(* CODESYS project ObjectOrientedProgramming.project
   Author: Manfred Werner
   Description: This example shows how OOP could be used to simplify the implementation of the management of different types of rooms.
      Start reading with the Interaces followed by the POU Building Manager.
   Title: Object Oriented Programming

Project tree, tasks and I/O mapping:
  Device : CODESYS Control Win V3 x64, 3S - Smart Software Solutions GmbH, version 3.5.15.0
    application BuildingApplication
      libraries: Util, 3.4.1.20 (System); Standard, * (System); CmpBitmapPool, * (System)
      task BuildingTask (cyclic, interval t#50ms, priority 1) calls BuildingManager
      Building_Objects/
        RoomFBs/
          function block RoomType3 [ST]: Operation_Daytime, SetTemperature, Operation_Nighttime, GetTemperature
          function block Roomtype1 [ST]: Operation_Daytime, SetLight, GetLight, Operation_Nighttime
          function block RoomType2 [ST]: SetLight
        function block CheckFB [CFC]
        Visualizations/
          visualisation Bulb
          visualisation Building
        global variables GlobalConstants
        program BuildingManager [ST]
        Interfaces/
          interface ITemp: SetTemperature, GetTemperature
          interface ILight: GetLight, SetLight
          interface IRoom: Operation_Nighttime, Operation_Daytime
      image pool ImagePool
      license
  libraries: VisuSymbols, 3.5.10.0 (System)
  text list GlobalTextList
  5ce3da45-db07-42e7-a21c-a00fff4ed8f6|C:\Users\a.werner\Documents\background.jpg
  00000000-0000-0000-0000-000000000000|C:\Users\m.lamp\Documents\license.txt
*)

// Device/BuildingApplication/Building_Objects/GlobalConstants
VAR_GLOBAL CONSTANT
	iNumberOfRooms:INT:=8;
END_VAR

// Device/BuildingApplication/Building_Objects/BuildingManager
PROGRAM BuildingManager
VAR
	(* define all rooms *)
	r1:RoomType1;		
	r2:RoomType3;
	r3:RoomType2;
	r4:RoomType3;
	r5:RoomType1;
	r6:RoomType3;
	r7:RoomType2;
	r8:RoomType1;
	(* Array of rooms simpilifies working with the building.*)
	Rooms: ARRAY [1..iNumberOfRooms] OF IRoom:=[r1,r2,r3,r4,r5,r6,r7,r8];
	CheckTimeOfDay: CheckFB; 	(* It's getting day? It's getting night? *)		
	xDusk: BOOL; (* nighttime *)
	xDawn:BOOL; (* daytime*)
	itfTemp: ITemp;
	xTemp: BOOL; (* Result of the Interface mapping.*) 
	i: INT;
END_VAR

(* Check if there is daytime or nighttime.*)
CheckTimeOfDay(xGetsDay=>xDawn,xGetsNight=>xDusk);
FOR i:=1 TO iNumberOfRooms DO
	IF xDawn THEN	(* Daytime*)
		Rooms[i].Operation_Daytime(); (* Disable the light and depending on the roomtype set the temperature. *)
	END_IF
	IF xDusk THEN	(* Nighttime *)
		Rooms[i].Operation_Nighttime(); (* Enable the light and depending on the roomtype set the temperature. *)
	END_IF
	
	(* If temperature is available for the Room, then set the temperature  --> RoomType3*)
	xTemp:=__QUERYINTERFACE(Rooms[i], itfTemp);
	IF xTemp AND i=6 THEN
		(* Now itfTemp has the address of Rooms[6] *)
		itfTemp.SetTemperature(35); (* The temperature of the Rooms[6] is set. *)
	END_IF
	
END_FOR

END_PROGRAM

// Device/BuildingApplication/Building_Objects/RoomFBs/RoomType3
(* Extended Room with an extra light and temperature. *)
FUNCTION_BLOCK RoomType3 EXTENDS Roomtype2 IMPLEMENTS ITemp
VAR_INPUT
END_VAR
VAR_OUTPUT
END_VAR
VAR
	iTemperature:INT;
END_VAR

(* This method overrides the inherited Operation_Daytime method from RoomType2. *)
METHOD Operation_Daytime : BOOL
VAR_INPUT
END_VAR
VAR
END_VAR
SUPER^.Operation_Daytime(); (* Disables the light.*)
SetTemperature(25); (* Additionally the temperature is set *)
END_METHOD

(* Implementation of the ITemp Interface *)
METHOD SetTemperature : BOOL
VAR_INPUT
	iNewTemperature:INT;
END_VAR
VAR
END_VAR
(* New temperature is set *)
iTemperature:=iNewTemperature;
END_METHOD

(* This method overrides the inherrited Operation_Nighttime method from RoomType2. *)
METHOD Operation_Nighttime : BOOL
VAR_INPUT
END_VAR
VAR
END_VAR
SUPER^.Operation_Nighttime(); (* Enables the light.*)
SetTemperature(15); (* Additionally the temperature is set *)
END_METHOD

(* Implementation of the ITemp Interface *)
METHOD GetTemperature : INT
VAR_INPUT
END_VAR
VAR
END_VAR
(* Get the temperature *)
GetTemperature:=iTemperature;
END_METHOD

END_FUNCTION_BLOCK

// Device/BuildingApplication/Building_Objects/RoomFBs/RoomType2
(* Extended Room with an extra light *)
FUNCTION_BLOCK RoomType2 EXTENDS Roomtype1
VAR_INPUT
END_VAR
VAR_OUTPUT
END_VAR
VAR
	bAdditionalLight:BOOL;
END_VAR

(* This method overrides the inherited SetLight method from RoomType1. *)
METHOD SetLight : BOOL
VAR_INPUT
	b:BOOL;
END_VAR
VAR
END_VAR
SUPER^.SetLight(b); (* Call the inherrited mehtod *)(* equal bLight:=b; *)
bAdditionalLight:=b;
END_METHOD

END_FUNCTION_BLOCK

// Device/BuildingApplication/Building_Objects/RoomFBs/Roomtype1
(* Simple room with only one light. *)	
FUNCTION_BLOCK Roomtype1 IMPLEMENTS IRoom, ILight
VAR_INPUT
END_VAR
VAR_OUTPUT
END_VAR
VAR
	bLight:BOOL;
END_VAR

(* Implementation of the IRoom Interface *)
METHOD Operation_Daytime : BOOL
VAR_INPUT
END_VAR
VAR
END_VAR
SetLight(FALSE); (* Disables the light *)
END_METHOD

(* Implementation of the ILight Interface *)
METHOD SetLight : BOOL
VAR_INPUT
	b:BOOL;
END_VAR
VAR
END_VAR
(* Set a new light value *)
bLight:=b;
END_METHOD

(* Implementation of the ILight Interface *)
METHOD GetLight : BOOL
VAR_INPUT
END_VAR
VAR
END_VAR
(* Returns the value of the light. *)
GetLight:=bLight;
END_METHOD

(* Implementation of the IRoom Interface *)
METHOD Operation_Nighttime : BOOL
VAR_INPUT
END_VAR
VAR
END_VAR
SetLight(TRUE); (* Enables the light *)
END_METHOD

END_FUNCTION_BLOCK

// Device/BuildingApplication/Building_Objects/Interfaces/IRoom
INTERFACE IRoom EXTENDS __system.IQueryInterface

METHOD Operation_Nighttime : BOOL
VAR_INPUT
END_VAR
VAR
END_VAR
END_METHOD

METHOD Operation_Daytime : BOOL
VAR_INPUT
END_VAR
VAR
END_VAR
END_METHOD

END_INTERFACE

// Device/BuildingApplication/Building_Objects/Interfaces/ILight
INTERFACE ILight

METHOD GetLight : BOOL
VAR_INPUT
END_VAR
VAR
END_VAR
END_METHOD

METHOD SetLight : BOOL
VAR_INPUT
	b:BOOL;
END_VAR
VAR
END_VAR
END_METHOD

END_INTERFACE

// Device/BuildingApplication/Building_Objects/Interfaces/ITemp
INTERFACE ITemp

METHOD SetTemperature : BOOL
VAR_INPUT
	iNewTemperature:INT;
END_VAR
VAR
END_VAR
END_METHOD

METHOD GetTemperature : INT
VAR_INPUT
END_VAR
VAR
END_VAR
END_METHOD

END_INTERFACE

// Device/BuildingApplication/Building_Objects/CheckFB
FUNCTION_BLOCK CheckFB
VAR_INPUT
END_VAR
VAR_OUTPUT
	xGetsNight:BOOL;
	xGetsDay:BOOL;
END_VAR
VAR
	blinking: BLINK;
	DayTrigger: R_TRIG;
	NightTrigger: F_TRIG;
END_VAR

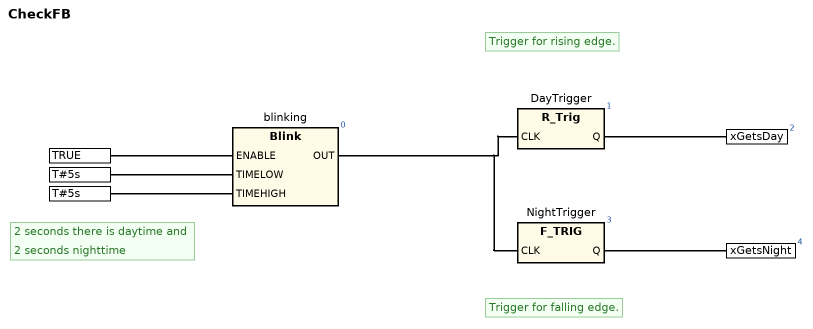
blinking(ENABLE := TRUE, TIMELOW := T#5s, TIMEHIGH := T#5s); // Blink
// Trigger for rising edge.
DayTrigger(CLK := blinking.OUT); // R_Trig
xGetsDay := DayTrigger.Q;
// 2 seconds there is daytime and
// 2 seconds nighttime
NightTrigger(CLK := blinking.OUT); // F_TRIG
// Trigger for falling edge.
xGetsNight := NightTrigger.Q;

END_FUNCTION_BLOCK

// Device/BuildingApplication/Building_Objects/Visualizations/Bulb
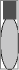
VISUALIZATION Bulb  // 19x70
VAR_INPUT
	bLight:BOOL;
END_VAR
    Ellipse (0,16 19x54), colour toggle: bLight
    Rectangle (3,0 13x19)
END_VISUALIZATION

// Device/BuildingApplication/Building_Objects/Visualizations/Building
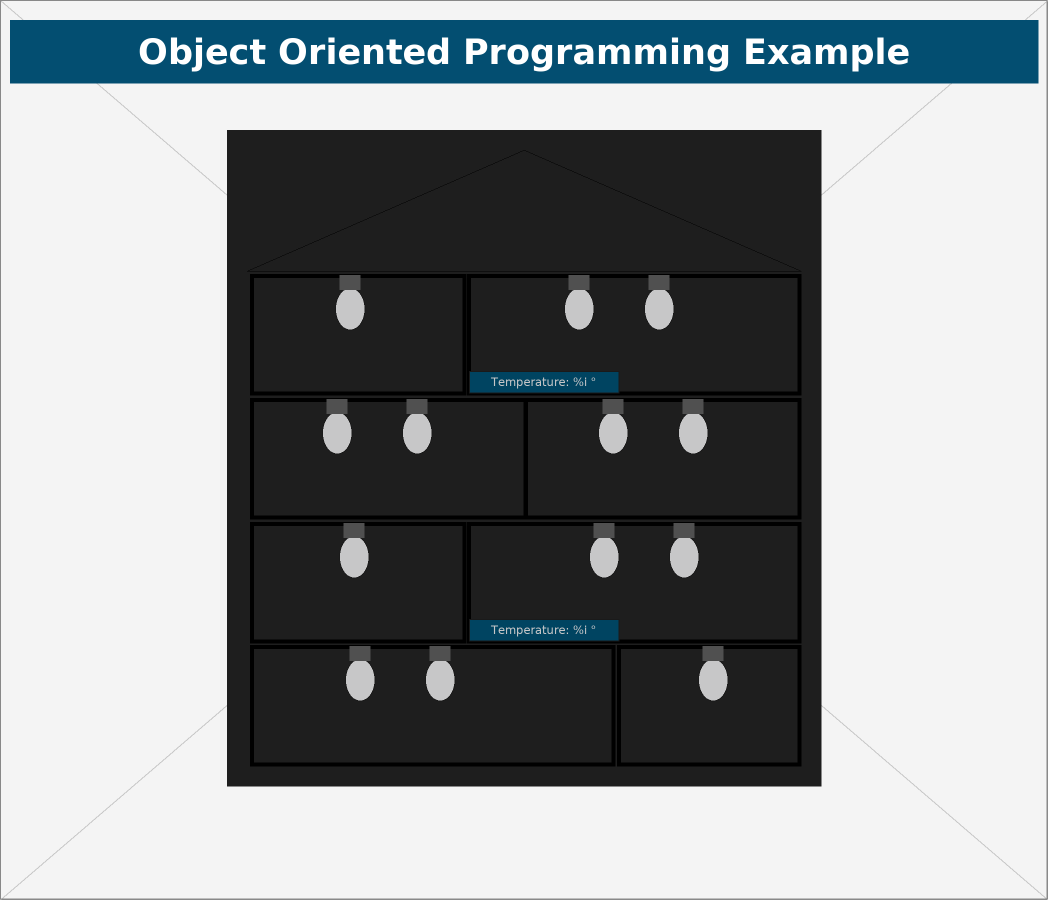
VISUALIZATION Building  // 1048x900
    Image (0,0 1048x900), image: ImagePool.background
    Rectangle (227,130 594x656)
    Rectangle (250,398 277x121)
    Polygon (524,150) (801,271) (247,271)
    Rectangle (250,274 216x121)
    Rectangle (467,274 334x121)
    Rectangle (469,371 150x22), "Temperature: %i °", text variable: BuildingManager.r2.iTemperature, colour toggle: BuildingManager.r2.iTemperature > 20
        p874137650: BuildingManager.r2.iTemperature * 2
    Rectangle (524,398 277x121)
    Rectangle (250,522 216x121)
    Rectangle (467,522 334x121)
    Rectangle (250,645 365x121)
    Rectangle (617,645 184x121)
    Frame (335,275 30x55)
        shows Bulb(bLight := BuildingManager.r1.bLight)
    Frame (564,275 30x55)
        shows Bulb(bLight := BuildingManager.r2.bLight)
    Frame (644,275 30x55)
        shows Bulb(bLight := BuildingManager.r2.bLight)
    Frame (322,399 30x55)
        shows Bulb(bLight := BuildingManager.r3.bLight)
    Frame (402,399 30x55)
        shows Bulb(bLight := BuildingManager.r3.bLight)
    Frame (598,399 30x55)
        shows Bulb(bLight := BuildingManager.r4.bLight)
    Frame (678,399 30x55)
        shows Bulb(bLight := BuildingManager.r4.bLight)
    Frame (345,646 30x55)
        shows Bulb(bLight := BuildingManager.r7.bLight)
    Frame (425,646 30x55)
        shows Bulb(bLight := BuildingManager.r7.bLight)
    Frame (589,523 30x55)
        shows Bulb(bLight := BuildingManager.r6.bLight)
    Frame (669,523 30x55)
        shows Bulb(bLight := BuildingManager.r6.bLight)
    Frame (339,523 30x55)
        shows Bulb(bLight := BuildingManager.r5.bLight)
    Frame (698,646 30x55)
        shows Bulb(bLight := BuildingManager.r8.bLight)
    Rectangle (469,619 150x22), "Temperature: %i °", text variable: BuildingManager.r6.iTemperature, colour toggle: BuildingManager.r6.iTemperature > 20
        p874137650: BuildingManager.r6.iTemperature * 2
    Rectangle (10,20 1028x63), "Object Oriented Programming Example"
END_VISUALIZATION
